Staubli VAL3: KIT.dtx

mdesc mNomSpeed
bool bSync
num nFileID
